{attribute 'qualified_only'}
{attribute 'strict'}
TYPE E_LeakLocation :
(
    NO_LEAK := 0,
    LOC1 := 1,
    LOC2 := 2,
    LOC3 := 4,
    LOC4 := 8,
    LOC5 := 16,
    LOC6 := 32
) BYTE;
END_TYPE

(* stored: Version 1.1.0.1, ProductVersion 3.1.4022.18
   DUT E_LeakLocation: Id {06f1d997-621d-4634-8016-7c31c5f73e8f} *)
